// TIA Portal V17 export
// export: Created 2024-08-20T13:36:59.3159366Z, ExportSetting WithDefaults, DisplayName Totally Integrated Automation Portal, DisplayVersion V17 Update 4, DisplayName TIA Portal Openness, DisplayVersion V17 Update 4, DisplayName TIA Portal Version Control Interface, DisplayVersion V17, DisplayName STEP 7 Professional, DisplayVersion V17 Update 4, DisplayName STEP 7 Safety, DisplayVersion V17, DisplayName WinCC Advanced, DisplayVersion V17 Update 4
FUNCTION_BLOCK "ROD4"   // FB200, LAD
TITLE = Rodízio de 4 grupos
{ S7_Optimized_Access := 'FALSE' }
VERSION : 0.1
// stored: AutoNumber false, IsIECCheckEnabled false, SetENOAutomatically false, UDAEnableTagReadback false
   VAR_INPUT
      G1OK : Bool;   // GRUPO EM CONDIÇÕES DE OPERAÇÃO
      G2OK : Bool;   // GRUPO EM CONDIÇÕES DE OPERAÇÃO
      G3OK : Bool;   // GRUPO EM CONDIÇÕES DE OPERAÇÃO
      G4OK : Bool;   // GRUPO EM CONDIÇÕES DE OPERAÇÃO
      G1L : Bool;   // GRUPO LIGADO
      G2L : Bool;   // GRUPO LIGADO
      G3L : Bool;   // GRUPO LIGADO
      G4L : Bool;   // GRUPO LIGADO
      TEROD : DInt;   // TEMPOPARA RODÍZIO DAS BOMBAS
      LIGP : Bool;   // LIGA BOMBA PRINCIPAL
      LIGC1 : Bool;   // LIGA BOMBA COMPLEMENTAR 1
      LIGC2 : Bool;   // LIGA BOMBA COMPLEMENTAR 2
      LIGC3 : Bool;   // LIGA BOMBA COMPLEMENTAR 3
      DESAB : Bool;   // DESABILITA FUNCIONAMENTO DOS GRUPOS
      T1S : Bool;   // PULSO A CADA 1 SEGUNDO
   END_VAR
   VAR_OUTPUT
      G1P : Bool;   // GRUPO 1 SELECIONADO COMO PRINCIPAL
      G2P : Bool;   // GRUPO 2 SELECIONADO COMO PRINCIPAL
      G3P : Bool;   // GRUPO 3 SELECIONADO COMO PRINCIPAL
      G4P : Bool;   // GRUPO 4 SELECIONADO COMO PRINCIPAL
      G1C1 : Bool;   // GRUPO 1 SELECIONADO COMO COMPLEMENTAR 1
      G2C1 : Bool;   // GRUPO 2 SELECIONADO COMO COMPLEMENTAR 1
      G3C1 : Bool;   // GRUPO 3 SELECIONADO COMO COMPLEMENTAR 1
      G4C1 : Bool;   // GRUPO 4 SELECIONADO COMO COMPLEMENTAR 1
      G1C2 : Bool;   // GRUPO 1 SELECIONADO COMO COMPLEMENTAR 2
      G2C2 : Bool;   // GRUPO 2 SELECIONADO COMO COMPLEMENTAR 2
      G3C2 : Bool;   // GRUPO 3 SELECIONADO COMO COMPLEMENTAR 3
      G4C2 : Bool;   // GRUPO 4 SELECIONADO COMO COMPLEMENTAR 4
      G1C3 : Bool;   // GRUPO 1 SELECIONADO COMO COMPLEMENTAR 3
      G2C3 : Bool;   // GRUPO 2 SELECIONADO COMO COMPLEMENTAR 3
      G3C3 : Bool;   // GRUPO 3 SELECIONADO COMO COMPLEMENTAR 3
      G4C3 : Bool;   // GRUPO 4 SELECIONADO COMO COMPLEMENTAR 3
      LG1 : Bool;   // LIGA GRUPO 1
      LG2 : Bool;   // LIGA GRUPO 2
      LG3 : Bool;   // LIGA GRUPO 3
      LG4 : Bool;   // LIGA GRUPO 4
   END_VAR
   VAR_IN_OUT
      TOG1P : DInt;   // TEMPO DE OPERAÇÃO GRUPO 1
      TOG2P : DInt;   // TEMPO DE OPERAÇÃO GRUPO 2
      TOG3P : DInt;   // TEMPO DE OPERAÇÃO GRUPO 3
      TOG4P : DInt;   // TEMPO DE OPERAÇÃO GRUPO 4
      TEOKG1 : Real;   // TEMPO OK GRUPO 1
      TEOKG2 : Real;   // TEMPO OK GRUPO 2
      TEOKG3 : Real;   // TEMPO OK GRUPO 3
      TEOKG4 : Real;   // TEMPO OK GRUPO 4
   END_VAR
   VAR DB_SPECIFIC
      GR1SELP : Bool;   // SELECIONADO COMO PRINCIPAL
      GR2SELP : Bool;   // SELECIONADO COMO PRINCIPAL
      GR3SELP : Bool;   // SELECIONADO COMO PRINCIPAL
      GR4SELP : Bool;   // SELECIONADO COMO PRINCIPAL
      GR1SELC1 : Bool;   // SELECIONADO COMO COMPLEMENTAR 1
      GR2SELC1 : Bool;   // SELECIONADO COMO COMPLEMENTAR 1
      GR3SELC1 : Bool;   // SELECIONADO COMO COMPLEMENTAR 1
      GR4SELC1 : Bool;   // SELECIONADO COMO COMPLEMENTAR 1
      GR1SELC2 : Bool;   // SELECIONADO COMO COMPLEMENTAR 2
      GR2SELC2 : Bool;   // SELECIONADO COMO COMPLEMENTAR 2
      GR3SELC2 : Bool;   // SELECIONADO COMO COMPLEMENTAR 2
      GR4SELC2 : Bool;   // SELECIONADO COMO COMPLEMENTAR 2
      GR1SELC3 : Bool;   // SELECIONADO COMO COMPLEMENTAR 3
      GR2SELC3 : Bool;   // SELECIONADO COMO COMPLEMENTAR 3
      GR3SELC3 : Bool;   // SELECIONADO COMO COMPLEMENTAR 3
      GR4SELC3 : Bool;   // SELECIONADO COMO COMPLEMENTAR 3
      PS1SG1 : Bool;   // AUXILIAR DE PULSO
      PS1SG2 : Bool;   // AUXILIAR DE PULSO
      PS1SG3 : Bool;   // AUXILIAR DE PULSO
      PS1SG4 : Bool;   // AUXILIAR DE PULSO
      PS1 : Bool;   // AUXILIAR DE PULSO
      PS2 : Bool;   // AUXILIAR DE PULSO
      PS3 : Bool;   // AUXILIAR DE PULSO
      PS4 : Bool;   // AUXILIAR DE PULSO
      FIMTEG1 : Bool;   // FIM DO TEMPO DE EXISTÊNCIA DO GRUPO 1
      FIMTEG2 : Bool;   // FIM DO TEMPO DE EXISTÊNCIA DO GRUPO 2
      FIMTEG3 : Bool;   // FIM DO TEMPO DE EXISTÊNCIA DO GRUPO 3
      FIMTEG4 : Bool;   // FIM DO TEMPO DE EXISTÊNCIA DO GRUPO 4
      SDESG1 : Bool;   // SOLICITAÇÃO DE DESLIGAMENTO
      SDESG2 : Bool;   // SOLICITAÇÃO DE DESLIGAMENTO
      SDESG3 : Bool;   // SOLICITAÇÃO DE DESLIGAMENTO
      SDESG4 : Bool;   // SOLICITAÇÃO DE DESLIGAMENTO
      GPL : Bool;   // GRUPO PRINCIPAL LIGADO
      GC1L : Bool;   // GRUPO COMPLEMENTAR 1 LIGADO
      GC2L : Bool;   // GRUPO COMPLEMENTAR 2 LIGADO
      GC3L : Bool;   // GRUPO COMPLEMENTAR 3 LIGADO
      SO_L : Bool;   // SOLICITAÇÃO DE PARTIDA
      SO_D : Bool;   // SOLICITAÇÃO DE DESLIGAMENTO
      RTEOKG1 : Bool;   // RESET TEMPO OK
      RTEOKG2 : Bool;   // RESET TEMPO OK
      RTEOKG3 : Bool;   // RESET TEMPO OK
      RTEOKG4 : Bool;   // RESET TEMPO OK
      TON1 { S7_SetPoint := 'True'} : TON_TIME;   // TEMPORIZADOR
      TON2 { S7_SetPoint := 'True'} : TON_TIME;   // TEMPORIZADOR
      TON3 { S7_SetPoint := 'True'} : TON_TIME;   // TEMPORIZADOR
      TON4 { S7_SetPoint := 'True'} : TON_TIME;   // TEMPORIZADOR
      TSDG1 { S7_SetPoint := 'True'} : TON_TIME;   // TEMPORIZADOR
      TSDG2 { S7_SetPoint := 'True'} : TON_TIME;   // TEMPORIZADOR
      TSDG3 { S7_SetPoint := 'True'} : TON_TIME;   // TEMPORIZADOR
      TSDG4 { S7_SetPoint := 'True'} : TON_TIME;   // TEMPORIZADOR
   END_VAR
   VAR_TEMP
      PRI12 : Bool;   // PRIORIDADE GRUPO 1
      PRI13 : Bool;   // PRIORIDADE GRUPO 1
      PRI14 : Bool;   // PRIORIDADE GRUPO 1
      PRI23 : Bool;   // PRIORIDADE GRUPO 2
      PRI24 : Bool;   // PRIORIDADE GRUPO 2
      PRI34 : Bool;   // PRIORIDADE GRUPO 3
      TMROD : Real;   // TEMPO DE RODIZIO
      NGS : Int;   // NÚMERO DE GRUPOS SOLICITADOS
      NGF : Int;   // NÚMERO DE GRUPOS FUNCIONANDO
      AUX01 : Int;   // AUXILIAR UTILIZADO NA LÓGICA
      AUX02 : Int;   // AUXILIAR UTILIZADO NA LÓGICA
      AUX03 : Int;   // AUXILIAR UTILIZADO NA LÓGICA
      AUX04 : Int;   // AUXILIAR UTILIZADO NA LÓGICA
      AUX05 : Bool;   // AUXILIAR UTILIZADO NA LÓGICA
      AUX06 : Bool;   // AUXILIAR UTILIZADO NA LÓGICA
      AUX07 : Bool;   // AUXILIAR UTILIZADO NA LÓGICA
      AUX08 : Bool;   // AUXILIAR UTILIZADO NA LÓGICA
      ETT1 : Time;   // EFETIVO DO TEMPORIZADOR
      ETT2 : Time;   // EFETIVO DO TEMPORIZADOR
      ETT3 : Time;   // EFETIVO DO TEMPORIZADOR
      ETT4 : Time;   // EFETIVO DO TEMPORIZADOR
      ETTSDG4 : Time;   // EFETIVO DO TEMPORIZADOR
      ETTSDG3 : Time;   // EFETIVO DO TEMPORIZADOR
      ETTSDG2 : Time;   // EFETIVO DO TEMPORIZADOR
      ETTSDG1 : Time;   // EFETIVO DO TEMPORIZADOR
   END_VAR
   VAR_TEMP   // added for the SCL form of the ladder/FBD networks
      _w1 : Bool;
   END_VAR
BEGIN

REGION Network 1: Tranforme em segundo o tempo de rodízio dos sopradores
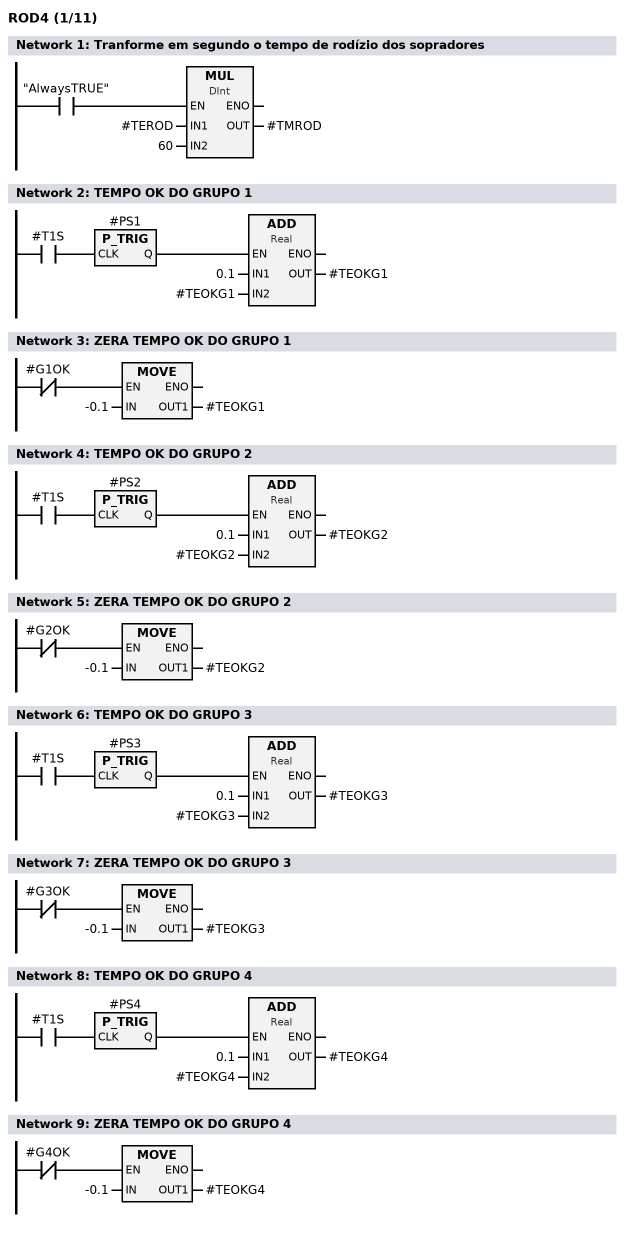
   RUNG wire#powerrail
      Contact( "AlwaysTRUE" )
      { S7_Templates := "SrcType := DInt"; S7_GenerateENO := "TRUE" } Mul(in1 := #TEROD, in2 := 60, out => #TMROD)
   END_RUNG
   // the same network as SCL:
   IF "AlwaysTRUE" THEN #TMROD := #TEROD * 60; END_IF;
END_REGION

REGION Network 2: TEMPO OK DO GRUPO 1
   RUNG wire#powerrail
      Contact( #T1S )
      P_Trig( #PS1 )
      { S7_Templates := "SrcType := Real"; S7_GenerateENO := "TRUE" } Add(in1 := 0.1, in2 := #TEOKG1, out => #TEOKG1)
   END_RUNG
   // the same network as SCL:
   #_w1 := #T1S AND NOT #PS1;   // rising edge
   #PS1 := #T1S;
   IF #_w1 THEN #TEOKG1 := 0.1 + #TEOKG1; END_IF;
END_REGION

REGION Network 3: ZERA TEMPO OK DO GRUPO 1
   RUNG wire#powerrail
      I_Contact( #G1OK )
      { S7_GenerateENO := "TRUE" } Move(in := -0.1, out1 => #TEOKG1)
   END_RUNG
   // the same network as SCL:
   IF NOT #G1OK THEN #TEOKG1 := -0.1; END_IF;
END_REGION

REGION Network 4: TEMPO OK DO GRUPO 2
   RUNG wire#powerrail
      Contact( #T1S )
      P_Trig( #PS2 )
      { S7_Templates := "SrcType := Real"; S7_GenerateENO := "TRUE" } Add(in1 := 0.1, in2 := #TEOKG2, out => #TEOKG2)
   END_RUNG
   // the same network as SCL:
   #_w1 := #T1S AND NOT #PS2;   // rising edge
   #PS2 := #T1S;
   IF #_w1 THEN #TEOKG2 := 0.1 + #TEOKG2; END_IF;
END_REGION

REGION Network 5: ZERA TEMPO OK DO GRUPO 2
   RUNG wire#powerrail
      I_Contact( #G2OK )
      { S7_GenerateENO := "TRUE" } Move(in := -0.1, out1 => #TEOKG2)
   END_RUNG
   // the same network as SCL:
   IF NOT #G2OK THEN #TEOKG2 := -0.1; END_IF;
END_REGION

REGION Network 6: TEMPO OK DO GRUPO 3
   RUNG wire#powerrail
      Contact( #T1S )
      P_Trig( #PS3 )
      { S7_Templates := "SrcType := Real"; S7_GenerateENO := "TRUE" } Add(in1 := 0.1, in2 := #TEOKG3, out => #TEOKG3)
   END_RUNG
   // the same network as SCL:
   #_w1 := #T1S AND NOT #PS3;   // rising edge
   #PS3 := #T1S;
   IF #_w1 THEN #TEOKG3 := 0.1 + #TEOKG3; END_IF;
END_REGION

REGION Network 7: ZERA TEMPO OK DO GRUPO 3
   RUNG wire#powerrail
      I_Contact( #G3OK )
      { S7_GenerateENO := "TRUE" } Move(in := -0.1, out1 => #TEOKG3)
   END_RUNG
   // the same network as SCL:
   IF NOT #G3OK THEN #TEOKG3 := -0.1; END_IF;
END_REGION

REGION Network 8: TEMPO OK DO GRUPO 4
   RUNG wire#powerrail
      Contact( #T1S )
      P_Trig( #PS4 )
      { S7_Templates := "SrcType := Real"; S7_GenerateENO := "TRUE" } Add(in1 := 0.1, in2 := #TEOKG4, out => #TEOKG4)
   END_RUNG
   // the same network as SCL:
   #_w1 := #T1S AND NOT #PS4;   // rising edge
   #PS4 := #T1S;
   IF #_w1 THEN #TEOKG4 := 0.1 + #TEOKG4; END_IF;
END_REGION

REGION Network 9: ZERA TEMPO OK DO GRUPO 4
   RUNG wire#powerrail
      I_Contact( #G4OK )
      { S7_GenerateENO := "TRUE" } Move(in := -0.1, out1 => #TEOKG4)
   END_RUNG
   // the same network as SCL:
   IF NOT #G4OK THEN #TEOKG4 := -0.1; END_IF;
END_REGION

REGION Network 10: DEFINIÇÇÃO DE PRIORIDADE DO GRUPO 1
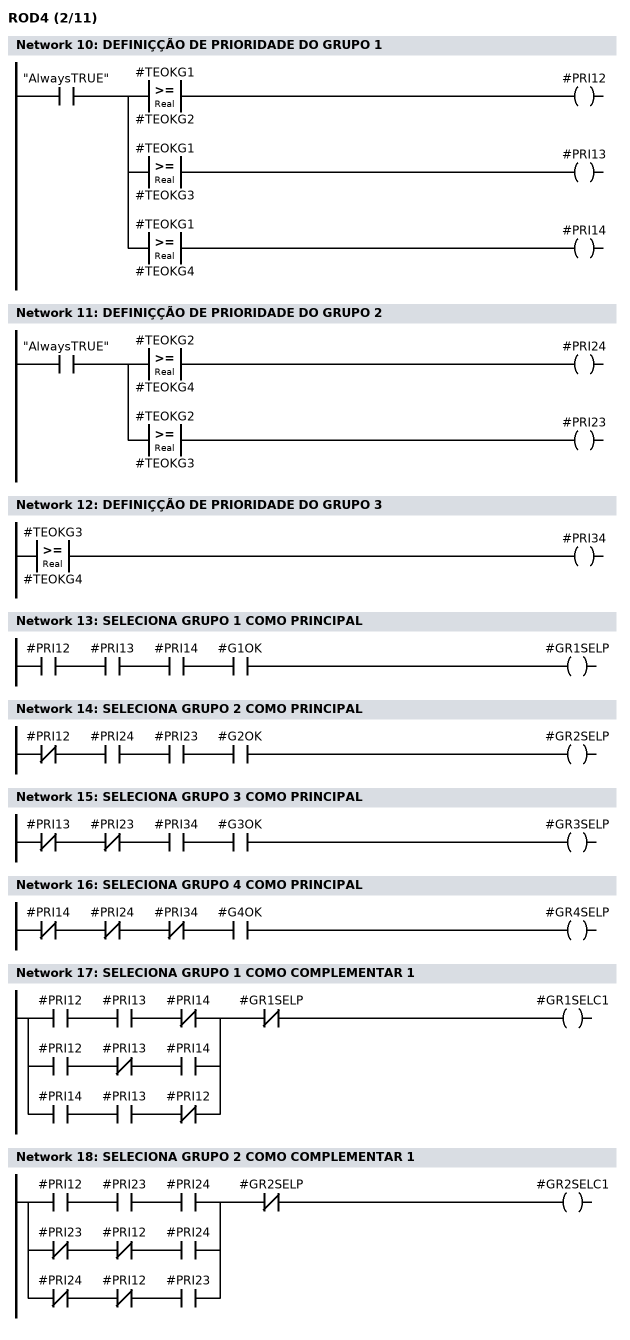
   RUNG wire#powerrail
      Contact( "AlwaysTRUE" )
      wire#w1
      { S7_Templates := "SrcType := Real" } GE_Contact(in1 := #TEOKG1, in2 := #TEOKG2)
      Coil( #PRI12 )
   END_RUNG
   RUNG wire#w1
      { S7_Templates := "SrcType := Real" } GE_Contact(in1 := #TEOKG1, in2 := #TEOKG3)
      Coil( #PRI13 )
   END_RUNG
   RUNG wire#w1
      { S7_Templates := "SrcType := Real" } GE_Contact(in1 := #TEOKG1, in2 := #TEOKG4)
      Coil( #PRI14 )
   END_RUNG
   // the same network as SCL:
   #PRI12 := "AlwaysTRUE" AND (#TEOKG1 >= #TEOKG2);
   #PRI13 := "AlwaysTRUE" AND (#TEOKG1 >= #TEOKG3);
   #PRI14 := "AlwaysTRUE" AND (#TEOKG1 >= #TEOKG4);
END_REGION

REGION Network 11: DEFINIÇÇÃO DE PRIORIDADE DO GRUPO 2
   RUNG wire#powerrail
      Contact( "AlwaysTRUE" )
      wire#w1
      { S7_Templates := "SrcType := Real" } GE_Contact(in1 := #TEOKG2, in2 := #TEOKG4)
      Coil( #PRI24 )
   END_RUNG
   RUNG wire#w1
      { S7_Templates := "SrcType := Real" } GE_Contact(in1 := #TEOKG2, in2 := #TEOKG3)
      Coil( #PRI23 )
   END_RUNG
   // the same network as SCL:
   #PRI24 := "AlwaysTRUE" AND (#TEOKG2 >= #TEOKG4);
   #PRI23 := "AlwaysTRUE" AND (#TEOKG2 >= #TEOKG3);
END_REGION

REGION Network 12: DEFINIÇÇÃO DE PRIORIDADE DO GRUPO 3
   RUNG wire#powerrail
      { S7_Templates := "SrcType := Real" } GE_Contact(in1 := #TEOKG3, in2 := #TEOKG4)
      Coil( #PRI34 )
   END_RUNG
   // the same network as SCL:
   #PRI34 := #TEOKG3 >= #TEOKG4;
END_REGION

REGION Network 13: SELECIONA GRUPO 1 COMO PRINCIPAL
   RUNG wire#powerrail
      Contact( #PRI12 )
      Contact( #PRI13 )
      Contact( #PRI14 )
      Contact( #G1OK )
      Coil( #GR1SELP )
   END_RUNG
   // the same network as SCL:
   #GR1SELP := #PRI12 AND #PRI13 AND #PRI14 AND #G1OK;
END_REGION

REGION Network 14: SELECIONA GRUPO 2 COMO PRINCIPAL
   RUNG wire#powerrail
      I_Contact( #PRI12 )
      Contact( #PRI24 )
      Contact( #PRI23 )
      Contact( #G2OK )
      Coil( #GR2SELP )
   END_RUNG
   // the same network as SCL:
   #GR2SELP := NOT #PRI12 AND #PRI24 AND #PRI23 AND #G2OK;
END_REGION

REGION Network 15: SELECIONA GRUPO 3 COMO PRINCIPAL
   RUNG wire#powerrail
      I_Contact( #PRI13 )
      I_Contact( #PRI23 )
      Contact( #PRI34 )
      Contact( #G3OK )
      Coil( #GR3SELP )
   END_RUNG
   // the same network as SCL:
   #GR3SELP := NOT #PRI13 AND NOT #PRI23 AND #PRI34 AND #G3OK;
END_REGION

REGION Network 16: SELECIONA GRUPO 4 COMO PRINCIPAL
   RUNG wire#powerrail
      I_Contact( #PRI14 )
      I_Contact( #PRI24 )
      I_Contact( #PRI34 )
      Contact( #G4OK )
      Coil( #GR4SELP )
   END_RUNG
   // the same network as SCL:
   #GR4SELP := NOT #PRI14 AND NOT #PRI24 AND NOT #PRI34 AND #G4OK;
END_REGION

REGION Network 17: SELECIONA GRUPO 1 COMO COMPLEMENTAR 1
   RUNG wire#powerrail
      Contact( #PRI12 )
      Contact( #PRI13 )
      I_Contact( #PRI14 )
      wire#w1
      I_Contact( #GR1SELP )
      Coil( #GR1SELC1 )
   END_RUNG
   RUNG wire#powerrail
      Contact( #PRI12 )
      I_Contact( #PRI13 )
      Contact( #PRI14 )
   END_RUNG wire#w1
   RUNG wire#powerrail
      Contact( #PRI14 )
      Contact( #PRI13 )
      I_Contact( #PRI12 )
   END_RUNG wire#w1
   // the same network as SCL:
   #GR1SELC1 := ((#PRI12 AND #PRI13 AND NOT #PRI14) OR (#PRI12 AND NOT #PRI13 AND #PRI14) OR (#PRI14 AND #PRI13 AND NOT #PRI12)) AND NOT #GR1SELP;
END_REGION

REGION Network 18: SELECIONA GRUPO 2 COMO COMPLEMENTAR 1
   RUNG wire#powerrail
      Contact( #PRI12 )
      Contact( #PRI23 )
      Contact( #PRI24 )
      wire#w1
      I_Contact( #GR2SELP )
      Coil( #GR2SELC1 )
   END_RUNG
   RUNG wire#powerrail
      I_Contact( #PRI23 )
      I_Contact( #PRI12 )
      Contact( #PRI24 )
   END_RUNG wire#w1
   RUNG wire#powerrail
      I_Contact( #PRI24 )
      I_Contact( #PRI12 )
      Contact( #PRI23 )
   END_RUNG wire#w1
   // the same network as SCL:
   #GR2SELC1 := ((#PRI12 AND #PRI23 AND #PRI24) OR (NOT #PRI23 AND NOT #PRI12 AND #PRI24) OR (NOT #PRI24 AND NOT #PRI12 AND #PRI23)) AND NOT #GR2SELP;
END_REGION

REGION Network 19: SELECIONA GRUPO 3 COMO COMPLEMENTAR 1
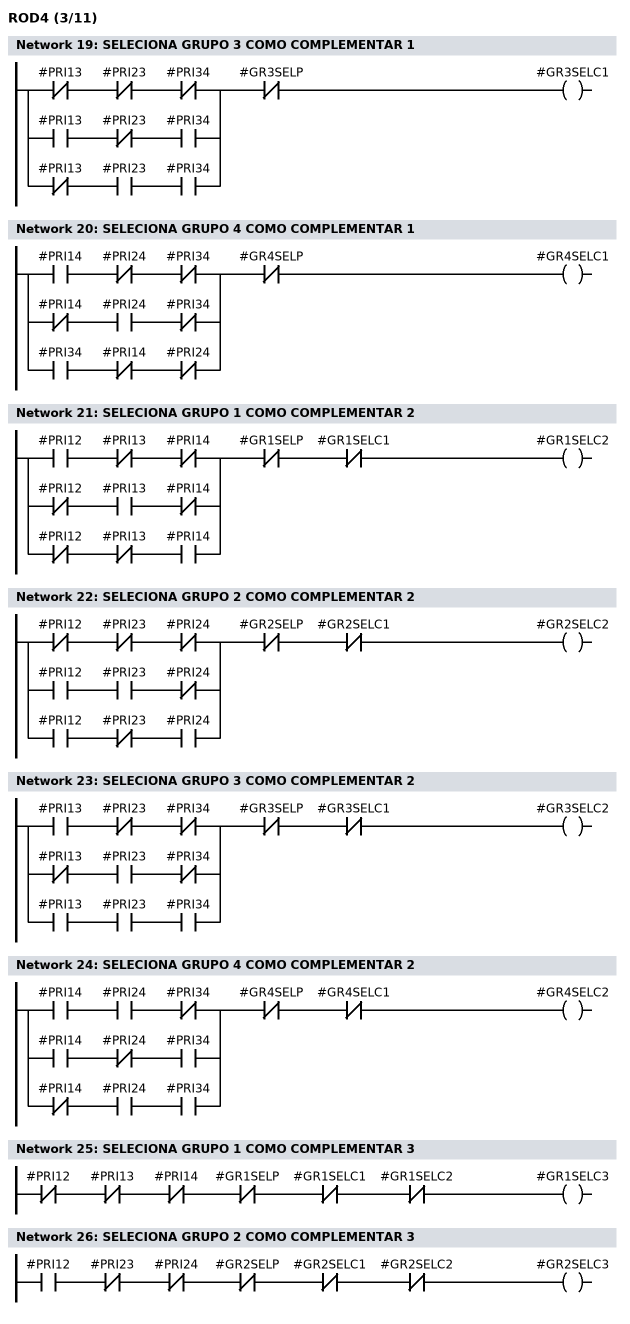
   RUNG wire#powerrail
      I_Contact( #PRI13 )
      I_Contact( #PRI23 )
      I_Contact( #PRI34 )
      wire#w1
      I_Contact( #GR3SELP )
      Coil( #GR3SELC1 )
   END_RUNG
   RUNG wire#powerrail
      Contact( #PRI13 )
      I_Contact( #PRI23 )
      Contact( #PRI34 )
   END_RUNG wire#w1
   RUNG wire#powerrail
      I_Contact( #PRI13 )
      Contact( #PRI23 )
      Contact( #PRI34 )
   END_RUNG wire#w1
   // the same network as SCL:
   #GR3SELC1 := ((NOT #PRI13 AND NOT #PRI23 AND NOT #PRI34) OR (#PRI13 AND NOT #PRI23 AND #PRI34) OR (NOT #PRI13 AND #PRI23 AND #PRI34)) AND NOT #GR3SELP;
END_REGION

REGION Network 20: SELECIONA GRUPO 4 COMO COMPLEMENTAR 1
   RUNG wire#powerrail
      Contact( #PRI14 )
      I_Contact( #PRI24 )
      I_Contact( #PRI34 )
      wire#w1
      I_Contact( #GR4SELP )
      Coil( #GR4SELC1 )
   END_RUNG
   RUNG wire#powerrail
      I_Contact( #PRI14 )
      Contact( #PRI24 )
      I_Contact( #PRI34 )
   END_RUNG wire#w1
   RUNG wire#powerrail
      Contact( #PRI34 )
      I_Contact( #PRI14 )
      I_Contact( #PRI24 )
   END_RUNG wire#w1
   // the same network as SCL:
   #GR4SELC1 := ((#PRI14 AND NOT #PRI24 AND NOT #PRI34) OR (NOT #PRI14 AND #PRI24 AND NOT #PRI34) OR (#PRI34 AND NOT #PRI14 AND NOT #PRI24)) AND NOT #GR4SELP;
END_REGION

REGION Network 21: SELECIONA GRUPO 1 COMO COMPLEMENTAR 2
   RUNG wire#powerrail
      Contact( #PRI12 )
      I_Contact( #PRI13 )
      I_Contact( #PRI14 )
      wire#w1
      I_Contact( #GR1SELP )
      I_Contact( #GR1SELC1 )
      Coil( #GR1SELC2 )
   END_RUNG
   RUNG wire#powerrail
      I_Contact( #PRI12 )
      Contact( #PRI13 )
      I_Contact( #PRI14 )
   END_RUNG wire#w1
   RUNG wire#powerrail
      I_Contact( #PRI12 )
      I_Contact( #PRI13 )
      Contact( #PRI14 )
   END_RUNG wire#w1
   // the same network as SCL:
   #GR1SELC2 := ((#PRI12 AND NOT #PRI13 AND NOT #PRI14) OR (NOT #PRI12 AND #PRI13 AND NOT #PRI14) OR (NOT #PRI12 AND NOT #PRI13 AND #PRI14)) AND NOT #GR1SELP AND NOT #GR1SELC1;
END_REGION

REGION Network 22: SELECIONA GRUPO 2 COMO COMPLEMENTAR 2
   RUNG wire#powerrail
      I_Contact( #PRI12 )
      I_Contact( #PRI23 )
      I_Contact( #PRI24 )
      wire#w1
      I_Contact( #GR2SELP )
      I_Contact( #GR2SELC1 )
      Coil( #GR2SELC2 )
   END_RUNG
   RUNG wire#powerrail
      Contact( #PRI12 )
      Contact( #PRI23 )
      I_Contact( #PRI24 )
   END_RUNG wire#w1
   RUNG wire#powerrail
      Contact( #PRI12 )
      I_Contact( #PRI23 )
      Contact( #PRI24 )
   END_RUNG wire#w1
   // the same network as SCL:
   #GR2SELC2 := ((NOT #PRI12 AND NOT #PRI23 AND NOT #PRI24) OR (#PRI12 AND #PRI23 AND NOT #PRI24) OR (#PRI12 AND NOT #PRI23 AND #PRI24)) AND NOT #GR2SELP AND NOT #GR2SELC1;
END_REGION

REGION Network 23: SELECIONA GRUPO 3 COMO COMPLEMENTAR 2
   RUNG wire#powerrail
      Contact( #PRI13 )
      I_Contact( #PRI23 )
      I_Contact( #PRI34 )
      wire#w1
      I_Contact( #GR3SELP )
      I_Contact( #GR3SELC1 )
      Coil( #GR3SELC2 )
   END_RUNG
   RUNG wire#powerrail
      I_Contact( #PRI13 )
      Contact( #PRI23 )
      I_Contact( #PRI34 )
   END_RUNG wire#w1
   RUNG wire#powerrail
      Contact( #PRI13 )
      Contact( #PRI23 )
      Contact( #PRI34 )
   END_RUNG wire#w1
   // the same network as SCL:
   #GR3SELC2 := ((#PRI13 AND NOT #PRI23 AND NOT #PRI34) OR (NOT #PRI13 AND #PRI23 AND NOT #PRI34) OR (#PRI13 AND #PRI23 AND #PRI34)) AND NOT #GR3SELP AND NOT #GR3SELC1;
END_REGION

REGION Network 24: SELECIONA GRUPO 4 COMO COMPLEMENTAR 2
   RUNG wire#powerrail
      Contact( #PRI14 )
      Contact( #PRI24 )
      I_Contact( #PRI34 )
      wire#w1
      I_Contact( #GR4SELP )
      I_Contact( #GR4SELC1 )
      Coil( #GR4SELC2 )
   END_RUNG
   RUNG wire#powerrail
      Contact( #PRI14 )
      I_Contact( #PRI24 )
      Contact( #PRI34 )
   END_RUNG wire#w1
   RUNG wire#powerrail
      I_Contact( #PRI14 )
      Contact( #PRI24 )
      Contact( #PRI34 )
   END_RUNG wire#w1
   // the same network as SCL:
   #GR4SELC2 := ((#PRI14 AND #PRI24 AND NOT #PRI34) OR (#PRI14 AND NOT #PRI24 AND #PRI34) OR (NOT #PRI14 AND #PRI24 AND #PRI34)) AND NOT #GR4SELP AND NOT #GR4SELC1;
END_REGION

REGION Network 25: SELECIONA GRUPO 1 COMO COMPLEMENTAR 3
   RUNG wire#powerrail
      I_Contact( #PRI12 )
      I_Contact( #PRI13 )
      I_Contact( #PRI14 )
      I_Contact( #GR1SELP )
      I_Contact( #GR1SELC1 )
      I_Contact( #GR1SELC2 )
      Coil( #GR1SELC3 )
   END_RUNG
   // the same network as SCL:
   #GR1SELC3 := NOT #PRI12 AND NOT #PRI13 AND NOT #PRI14 AND NOT #GR1SELP AND NOT #GR1SELC1 AND NOT #GR1SELC2;
END_REGION

REGION Network 26: SELECIONA GRUPO 2 COMO COMPLEMENTAR 3
   RUNG wire#powerrail
      Contact( #PRI12 )
      I_Contact( #PRI23 )
      I_Contact( #PRI24 )
      I_Contact( #GR2SELP )
      I_Contact( #GR2SELC1 )
      I_Contact( #GR2SELC2 )
      Coil( #GR2SELC3 )
   END_RUNG
   // the same network as SCL:
   #GR2SELC3 := #PRI12 AND NOT #PRI23 AND NOT #PRI24 AND NOT #GR2SELP AND NOT #GR2SELC1 AND NOT #GR2SELC2;
END_REGION

REGION Network 27: SELECIONA GRUPO 3 COMO COMPLEMENTAR 3
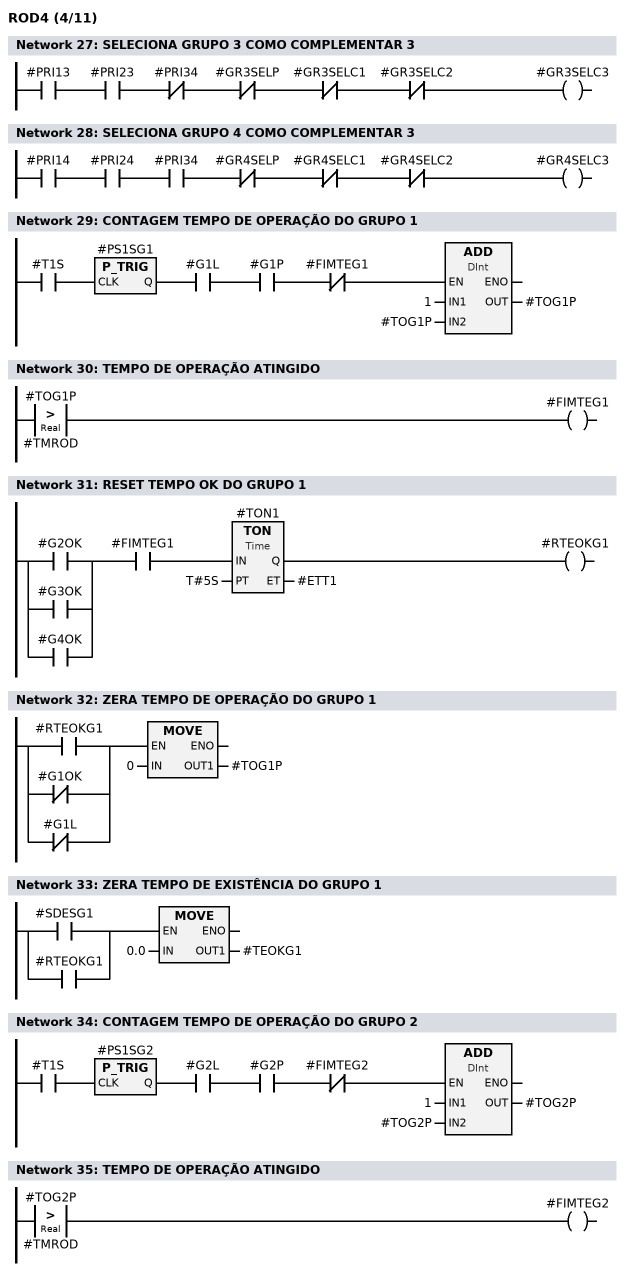
   RUNG wire#powerrail
      Contact( #PRI13 )
      Contact( #PRI23 )
      I_Contact( #PRI34 )
      I_Contact( #GR3SELP )
      I_Contact( #GR3SELC1 )
      I_Contact( #GR3SELC2 )
      Coil( #GR3SELC3 )
   END_RUNG
   // the same network as SCL:
   #GR3SELC3 := #PRI13 AND #PRI23 AND NOT #PRI34 AND NOT #GR3SELP AND NOT #GR3SELC1 AND NOT #GR3SELC2;
END_REGION

REGION Network 28: SELECIONA GRUPO 4 COMO COMPLEMENTAR 3
   RUNG wire#powerrail
      Contact( #PRI14 )
      Contact( #PRI24 )
      Contact( #PRI34 )
      I_Contact( #GR4SELP )
      I_Contact( #GR4SELC1 )
      I_Contact( #GR4SELC2 )
      Coil( #GR4SELC3 )
   END_RUNG
   // the same network as SCL:
   #GR4SELC3 := #PRI14 AND #PRI24 AND #PRI34 AND NOT #GR4SELP AND NOT #GR4SELC1 AND NOT #GR4SELC2;
END_REGION

REGION Network 29: CONTAGEM TEMPO DE OPERAÇÃO DO GRUPO 1
   RUNG wire#powerrail
      Contact( #T1S )
      P_Trig( #PS1SG1 )
      Contact( #G1L )
      Contact( #G1P )
      I_Contact( #FIMTEG1 )
      { S7_Templates := "SrcType := DInt"; S7_GenerateENO := "TRUE" } Add(in1 := 1, in2 := #TOG1P, out => #TOG1P)
   END_RUNG
   // the same network as SCL:
   #_w1 := #T1S AND NOT #PS1SG1;   // rising edge
   #PS1SG1 := #T1S;
   IF #_w1 AND #G1L AND #G1P AND NOT #FIMTEG1 THEN #TOG1P := 1 + #TOG1P; END_IF;
END_REGION

REGION Network 30: TEMPO DE OPERAÇÃO ATINGIDO
   RUNG wire#powerrail
      { S7_Templates := "SrcType := Real" } GT_Contact(in1 := #TOG1P, in2 := #TMROD)
      Coil( #FIMTEG1 )
   END_RUNG
   // the same network as SCL:
   #FIMTEG1 := #TOG1P > #TMROD;
END_REGION

REGION Network 31: RESET TEMPO OK DO GRUPO 1
   RUNG wire#powerrail
      Contact( #G2OK )
      wire#w1
      Contact( #FIMTEG1 )
      { S7_Templates := "time_type := Time" } #TON1.TON(pt := T#5S, et => #ETT1)
      Coil( #RTEOKG1 )
   END_RUNG
   RUNG wire#powerrail
      Contact( #G3OK )
   END_RUNG wire#w1
   RUNG wire#powerrail
      Contact( #G4OK )
   END_RUNG wire#w1
   // the same network as SCL:
   #TON1(IN := (#G2OK OR #G3OK OR #G4OK) AND #FIMTEG1, PT := T#5S, ET => #ETT1);   // TON
   #RTEOKG1 := #TON1.Q;
END_REGION

REGION Network 32: ZERA TEMPO DE OPERAÇÃO DO GRUPO 1
   RUNG wire#powerrail
      Contact( #RTEOKG1 )
      wire#w1
      { S7_GenerateENO := "TRUE" } Move(in := 0, out1 => #TOG1P)
   END_RUNG
   RUNG wire#powerrail
      I_Contact( #G1OK )
   END_RUNG wire#w1
   RUNG wire#powerrail
      I_Contact( #G1L )
   END_RUNG wire#w1
   // the same network as SCL:
   IF #RTEOKG1 OR NOT #G1OK OR NOT #G1L THEN #TOG1P := 0; END_IF;
END_REGION

REGION Network 33: ZERA TEMPO DE EXISTÊNCIA DO GRUPO 1
   RUNG wire#powerrail
      Contact( #SDESG1 )
      wire#w1
      { S7_GenerateENO := "TRUE" } Move(in := 0.0, out1 => #TEOKG1)
   END_RUNG
   RUNG wire#powerrail
      Contact( #RTEOKG1 )
   END_RUNG wire#w1
   // the same network as SCL:
   IF #SDESG1 OR #RTEOKG1 THEN #TEOKG1 := 0.0; END_IF;
END_REGION

REGION Network 34: CONTAGEM TEMPO DE OPERAÇÃO DO GRUPO 2
   RUNG wire#powerrail
      Contact( #T1S )
      P_Trig( #PS1SG2 )
      Contact( #G2L )
      Contact( #G2P )
      I_Contact( #FIMTEG2 )
      { S7_Templates := "SrcType := DInt"; S7_GenerateENO := "TRUE" } Add(in1 := 1, in2 := #TOG2P, out => #TOG2P)
   END_RUNG
   // the same network as SCL:
   #_w1 := #T1S AND NOT #PS1SG2;   // rising edge
   #PS1SG2 := #T1S;
   IF #_w1 AND #G2L AND #G2P AND NOT #FIMTEG2 THEN #TOG2P := 1 + #TOG2P; END_IF;
END_REGION

REGION Network 35: TEMPO DE OPERAÇÃO ATINGIDO
   RUNG wire#powerrail
      { S7_Templates := "SrcType := Real" } GT_Contact(in1 := #TOG2P, in2 := #TMROD)
      Coil( #FIMTEG2 )
   END_RUNG
   // the same network as SCL:
   #FIMTEG2 := #TOG2P > #TMROD;
END_REGION

REGION Network 36: RESET TEMPO OK DO GRUPO 2
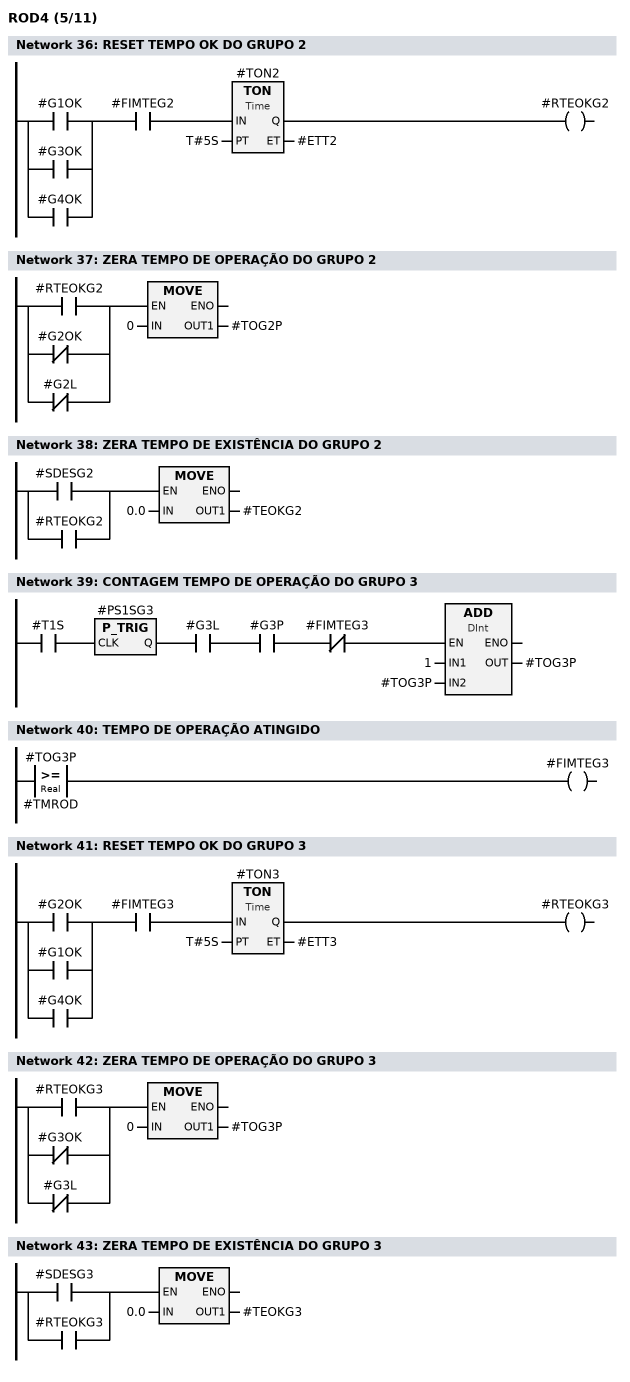
   RUNG wire#powerrail
      Contact( #G1OK )
      wire#w1
      Contact( #FIMTEG2 )
      { S7_Templates := "time_type := Time" } #TON2.TON(pt := T#5S, et => #ETT2)
      Coil( #RTEOKG2 )
   END_RUNG
   RUNG wire#powerrail
      Contact( #G3OK )
   END_RUNG wire#w1
   RUNG wire#powerrail
      Contact( #G4OK )
   END_RUNG wire#w1
   // the same network as SCL:
   #TON2(IN := (#G1OK OR #G3OK OR #G4OK) AND #FIMTEG2, PT := T#5S, ET => #ETT2);   // TON
   #RTEOKG2 := #TON2.Q;
END_REGION

REGION Network 37: ZERA TEMPO DE OPERAÇÃO DO GRUPO 2
   RUNG wire#powerrail
      Contact( #RTEOKG2 )
      wire#w1
      { S7_GenerateENO := "TRUE" } Move(in := 0, out1 => #TOG2P)
   END_RUNG
   RUNG wire#powerrail
      I_Contact( #G2OK )
   END_RUNG wire#w1
   RUNG wire#powerrail
      I_Contact( #G2L )
   END_RUNG wire#w1
   // the same network as SCL:
   IF #RTEOKG2 OR NOT #G2OK OR NOT #G2L THEN #TOG2P := 0; END_IF;
END_REGION

REGION Network 38: ZERA TEMPO DE EXISTÊNCIA DO GRUPO 2
   RUNG wire#powerrail
      Contact( #SDESG2 )
      wire#w1
      { S7_GenerateENO := "TRUE" } Move(in := 0.0, out1 => #TEOKG2)
   END_RUNG
   RUNG wire#powerrail
      Contact( #RTEOKG2 )
   END_RUNG wire#w1
   // the same network as SCL:
   IF #SDESG2 OR #RTEOKG2 THEN #TEOKG2 := 0.0; END_IF;
END_REGION

REGION Network 39: CONTAGEM TEMPO DE OPERAÇÃO DO GRUPO 3
   RUNG wire#powerrail
      Contact( #T1S )
      P_Trig( #PS1SG3 )
      Contact( #G3L )
      Contact( #G3P )
      I_Contact( #FIMTEG3 )
      { S7_Templates := "SrcType := DInt"; S7_GenerateENO := "TRUE" } Add(in1 := 1, in2 := #TOG3P, out => #TOG3P)
   END_RUNG
   // the same network as SCL:
   #_w1 := #T1S AND NOT #PS1SG3;   // rising edge
   #PS1SG3 := #T1S;
   IF #_w1 AND #G3L AND #G3P AND NOT #FIMTEG3 THEN #TOG3P := 1 + #TOG3P; END_IF;
END_REGION

REGION Network 40: TEMPO DE OPERAÇÃO ATINGIDO
   RUNG wire#powerrail
      { S7_Templates := "SrcType := Real" } GE_Contact(in1 := #TOG3P, in2 := #TMROD)
      Coil( #FIMTEG3 )
   END_RUNG
   // the same network as SCL:
   #FIMTEG3 := #TOG3P >= #TMROD;
END_REGION

REGION Network 41: RESET TEMPO OK DO GRUPO 3
   RUNG wire#powerrail
      Contact( #G2OK )
      wire#w1
      Contact( #FIMTEG3 )
      { S7_Templates := "time_type := Time" } #TON3.TON(pt := T#5S, et => #ETT3)
      Coil( #RTEOKG3 )
   END_RUNG
   RUNG wire#powerrail
      Contact( #G1OK )
   END_RUNG wire#w1
   RUNG wire#powerrail
      Contact( #G4OK )
   END_RUNG wire#w1
   // the same network as SCL:
   #TON3(IN := (#G2OK OR #G1OK OR #G4OK) AND #FIMTEG3, PT := T#5S, ET => #ETT3);   // TON
   #RTEOKG3 := #TON3.Q;
END_REGION

REGION Network 42: ZERA TEMPO DE OPERAÇÃO DO GRUPO 3
   RUNG wire#powerrail
      Contact( #RTEOKG3 )
      wire#w1
      { S7_GenerateENO := "TRUE" } Move(in := 0, out1 => #TOG3P)
   END_RUNG
   RUNG wire#powerrail
      I_Contact( #G3OK )
   END_RUNG wire#w1
   RUNG wire#powerrail
      I_Contact( #G3L )
   END_RUNG wire#w1
   // the same network as SCL:
   IF #RTEOKG3 OR NOT #G3OK OR NOT #G3L THEN #TOG3P := 0; END_IF;
END_REGION

REGION Network 43: ZERA TEMPO DE EXISTÊNCIA DO GRUPO 3
   RUNG wire#powerrail
      Contact( #SDESG3 )
      wire#w1
      { S7_GenerateENO := "TRUE" } Move(in := 0.0, out1 => #TEOKG3)
   END_RUNG
   RUNG wire#powerrail
      Contact( #RTEOKG3 )
   END_RUNG wire#w1
   // the same network as SCL:
   IF #SDESG3 OR #RTEOKG3 THEN #TEOKG3 := 0.0; END_IF;
END_REGION

REGION Network 44: CONTAGEM TEMPO DE OPERAÇÃO DO GRUPO 4
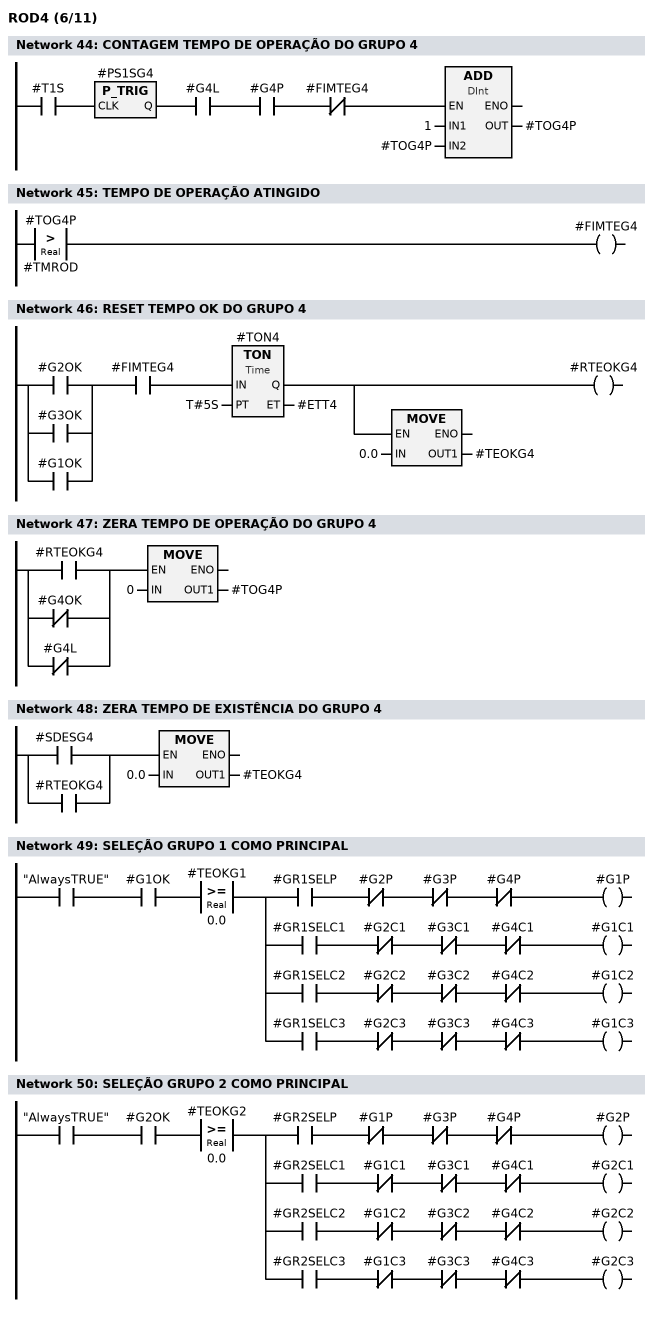
   RUNG wire#powerrail
      Contact( #T1S )
      P_Trig( #PS1SG4 )
      Contact( #G4L )
      Contact( #G4P )
      I_Contact( #FIMTEG4 )
      { S7_Templates := "SrcType := DInt"; S7_GenerateENO := "TRUE" } Add(in1 := 1, in2 := #TOG4P, out => #TOG4P)
   END_RUNG
   // the same network as SCL:
   #_w1 := #T1S AND NOT #PS1SG4;   // rising edge
   #PS1SG4 := #T1S;
   IF #_w1 AND #G4L AND #G4P AND NOT #FIMTEG4 THEN #TOG4P := 1 + #TOG4P; END_IF;
END_REGION

REGION Network 45: TEMPO DE OPERAÇÃO ATINGIDO
   RUNG wire#powerrail
      { S7_Templates := "SrcType := Real" } GT_Contact(in1 := #TOG4P, in2 := #TMROD)
      Coil( #FIMTEG4 )
   END_RUNG
   // the same network as SCL:
   #FIMTEG4 := #TOG4P > #TMROD;
END_REGION

REGION Network 46: RESET TEMPO OK DO GRUPO 4
   RUNG wire#powerrail
      Contact( #G2OK )
      wire#w1
      Contact( #FIMTEG4 )
      { S7_Templates := "time_type := Time" } #TON4.TON(pt := T#5S, et => #ETT4)
      wire#w2
      Coil( #RTEOKG4 )
   END_RUNG
   RUNG wire#powerrail
      Contact( #G3OK )
   END_RUNG wire#w1
   RUNG wire#powerrail
      Contact( #G1OK )
   END_RUNG wire#w1
   RUNG wire#w2
      { S7_GenerateENO := "TRUE" } Move(in := 0.0, out1 => #TEOKG4)
   END_RUNG
   // the same network as SCL:
   #TON4(IN := (#G2OK OR #G3OK OR #G1OK) AND #FIMTEG4, PT := T#5S, ET => #ETT4);   // TON
   #RTEOKG4 := #TON4.Q;
   IF #TON4.Q THEN #TEOKG4 := 0.0; END_IF;
END_REGION

REGION Network 47: ZERA TEMPO DE OPERAÇÃO DO GRUPO 4
   RUNG wire#powerrail
      Contact( #RTEOKG4 )
      wire#w1
      { S7_GenerateENO := "TRUE" } Move(in := 0, out1 => #TOG4P)
   END_RUNG
   RUNG wire#powerrail
      I_Contact( #G4OK )
   END_RUNG wire#w1
   RUNG wire#powerrail
      I_Contact( #G4L )
   END_RUNG wire#w1
   // the same network as SCL:
   IF #RTEOKG4 OR NOT #G4OK OR NOT #G4L THEN #TOG4P := 0; END_IF;
END_REGION

REGION Network 48: ZERA TEMPO DE EXISTÊNCIA DO GRUPO 4
   RUNG wire#powerrail
      Contact( #SDESG4 )
      wire#w1
      { S7_GenerateENO := "TRUE" } Move(in := 0.0, out1 => #TEOKG4)
   END_RUNG
   RUNG wire#powerrail
      Contact( #RTEOKG4 )
   END_RUNG wire#w1
   // the same network as SCL:
   IF #SDESG4 OR #RTEOKG4 THEN #TEOKG4 := 0.0; END_IF;
END_REGION

REGION Network 49: SELEÇÃO GRUPO 1 COMO PRINCIPAL
   RUNG wire#powerrail
      Contact( "AlwaysTRUE" )
      Contact( #G1OK )
      { S7_Templates := "SrcType := Real" } GE_Contact(in1 := #TEOKG1, in2 := 0.0)
      wire#w1
      Contact( #GR1SELP )
      I_Contact( #G2P )
      I_Contact( #G3P )
      I_Contact( #G4P )
      Coil( #G1P )
   END_RUNG
   RUNG wire#w1
      Contact( #GR1SELC1 )
      I_Contact( #G2C1 )
      I_Contact( #G3C1 )
      I_Contact( #G4C1 )
      Coil( #G1C1 )
   END_RUNG
   RUNG wire#w1
      Contact( #GR1SELC2 )
      I_Contact( #G2C2 )
      I_Contact( #G3C2 )
      I_Contact( #G4C2 )
      Coil( #G1C2 )
   END_RUNG
   RUNG wire#w1
      Contact( #GR1SELC3 )
      I_Contact( #G2C3 )
      I_Contact( #G3C3 )
      I_Contact( #G4C3 )
      Coil( #G1C3 )
   END_RUNG
   // the same network as SCL:
   #_w1 := "AlwaysTRUE" AND #G1OK AND (#TEOKG1 >= 0.0);
   #G1P := #_w1 AND #GR1SELP AND NOT #G2P AND NOT #G3P AND NOT #G4P;
   #G1C1 := #_w1 AND #GR1SELC1 AND NOT #G2C1 AND NOT #G3C1 AND NOT #G4C1;
   #G1C2 := #_w1 AND #GR1SELC2 AND NOT #G2C2 AND NOT #G3C2 AND NOT #G4C2;
   #G1C3 := #_w1 AND #GR1SELC3 AND NOT #G2C3 AND NOT #G3C3 AND NOT #G4C3;
END_REGION

REGION Network 50: SELEÇÃO GRUPO 2 COMO PRINCIPAL
   RUNG wire#powerrail
      Contact( "AlwaysTRUE" )
      Contact( #G2OK )
      { S7_Templates := "SrcType := Real" } GE_Contact(in1 := #TEOKG2, in2 := 0.0)
      wire#w1
      Contact( #GR2SELP )
      I_Contact( #G1P )
      I_Contact( #G3P )
      I_Contact( #G4P )
      Coil( #G2P )
   END_RUNG
   RUNG wire#w1
      Contact( #GR2SELC1 )
      I_Contact( #G1C1 )
      I_Contact( #G3C1 )
      I_Contact( #G4C1 )
      Coil( #G2C1 )
   END_RUNG
   RUNG wire#w1
      Contact( #GR2SELC2 )
      I_Contact( #G1C2 )
      I_Contact( #G3C2 )
      I_Contact( #G4C2 )
      Coil( #G2C2 )
   END_RUNG
   RUNG wire#w1
      Contact( #GR2SELC3 )
      I_Contact( #G1C3 )
      I_Contact( #G3C3 )
      I_Contact( #G4C3 )
      Coil( #G2C3 )
   END_RUNG
   // the same network as SCL:
   #_w1 := "AlwaysTRUE" AND #G2OK AND (#TEOKG2 >= 0.0);
   #G2P := #_w1 AND #GR2SELP AND NOT #G1P AND NOT #G3P AND NOT #G4P;
   #G2C1 := #_w1 AND #GR2SELC1 AND NOT #G1C1 AND NOT #G3C1 AND NOT #G4C1;
   #G2C2 := #_w1 AND #GR2SELC2 AND NOT #G1C2 AND NOT #G3C2 AND NOT #G4C2;
   #G2C3 := #_w1 AND #GR2SELC3 AND NOT #G1C3 AND NOT #G3C3 AND NOT #G4C3;
END_REGION

REGION Network 51: SELEÇÃO GRUPO 3 COMO PRINCIPAL
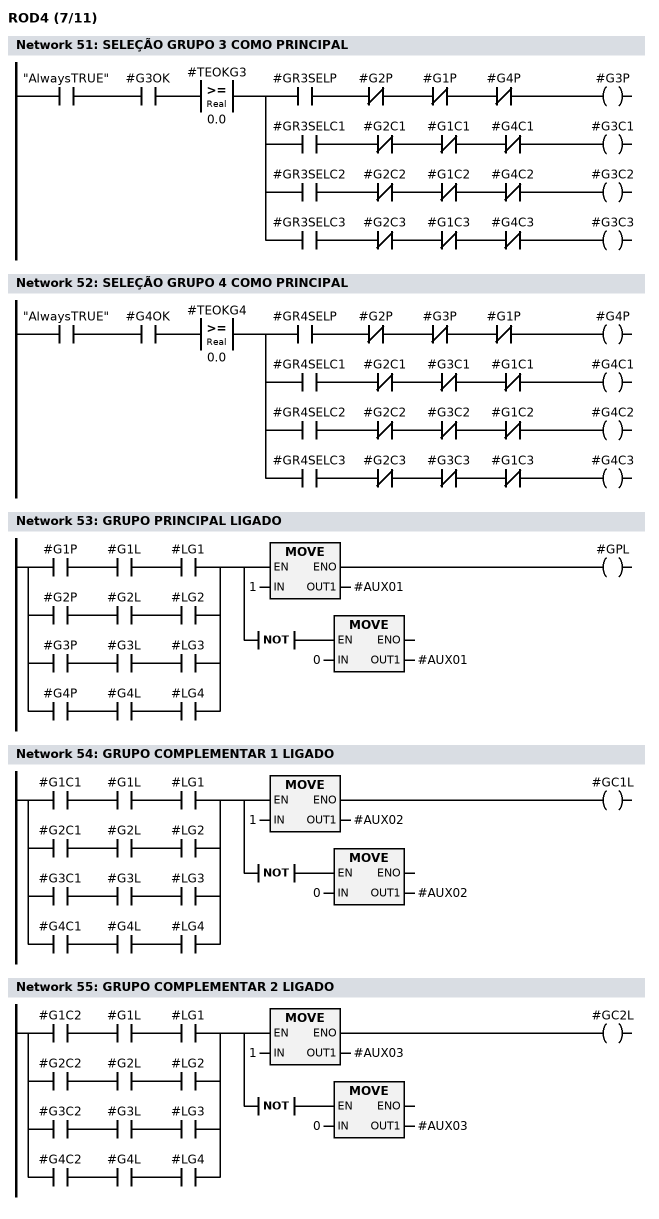
   RUNG wire#powerrail
      Contact( "AlwaysTRUE" )
      Contact( #G3OK )
      { S7_Templates := "SrcType := Real" } GE_Contact(in1 := #TEOKG3, in2 := 0.0)
      wire#w1
      Contact( #GR3SELP )
      I_Contact( #G2P )
      I_Contact( #G1P )
      I_Contact( #G4P )
      Coil( #G3P )
   END_RUNG
   RUNG wire#w1
      Contact( #GR3SELC1 )
      I_Contact( #G2C1 )
      I_Contact( #G1C1 )
      I_Contact( #G4C1 )
      Coil( #G3C1 )
   END_RUNG
   RUNG wire#w1
      Contact( #GR3SELC2 )
      I_Contact( #G2C2 )
      I_Contact( #G1C2 )
      I_Contact( #G4C2 )
      Coil( #G3C2 )
   END_RUNG
   RUNG wire#w1
      Contact( #GR3SELC3 )
      I_Contact( #G2C3 )
      I_Contact( #G1C3 )
      I_Contact( #G4C3 )
      Coil( #G3C3 )
   END_RUNG
   // the same network as SCL:
   #_w1 := "AlwaysTRUE" AND #G3OK AND (#TEOKG3 >= 0.0);
   #G3P := #_w1 AND #GR3SELP AND NOT #G2P AND NOT #G1P AND NOT #G4P;
   #G3C1 := #_w1 AND #GR3SELC1 AND NOT #G2C1 AND NOT #G1C1 AND NOT #G4C1;
   #G3C2 := #_w1 AND #GR3SELC2 AND NOT #G2C2 AND NOT #G1C2 AND NOT #G4C2;
   #G3C3 := #_w1 AND #GR3SELC3 AND NOT #G2C3 AND NOT #G1C3 AND NOT #G4C3;
END_REGION

REGION Network 52: SELEÇÃO GRUPO 4 COMO PRINCIPAL
   RUNG wire#powerrail
      Contact( "AlwaysTRUE" )
      Contact( #G4OK )
      { S7_Templates := "SrcType := Real" } GE_Contact(in1 := #TEOKG4, in2 := 0.0)
      wire#w1
      Contact( #GR4SELP )
      I_Contact( #G2P )
      I_Contact( #G3P )
      I_Contact( #G1P )
      Coil( #G4P )
   END_RUNG
   RUNG wire#w1
      Contact( #GR4SELC1 )
      I_Contact( #G2C1 )
      I_Contact( #G3C1 )
      I_Contact( #G1C1 )
      Coil( #G4C1 )
   END_RUNG
   RUNG wire#w1
      Contact( #GR4SELC2 )
      I_Contact( #G2C2 )
      I_Contact( #G3C2 )
      I_Contact( #G1C2 )
      Coil( #G4C2 )
   END_RUNG
   RUNG wire#w1
      Contact( #GR4SELC3 )
      I_Contact( #G2C3 )
      I_Contact( #G3C3 )
      I_Contact( #G1C3 )
      Coil( #G4C3 )
   END_RUNG
   // the same network as SCL:
   #_w1 := "AlwaysTRUE" AND #G4OK AND (#TEOKG4 >= 0.0);
   #G4P := #_w1 AND #GR4SELP AND NOT #G2P AND NOT #G3P AND NOT #G1P;
   #G4C1 := #_w1 AND #GR4SELC1 AND NOT #G2C1 AND NOT #G3C1 AND NOT #G1C1;
   #G4C2 := #_w1 AND #GR4SELC2 AND NOT #G2C2 AND NOT #G3C2 AND NOT #G1C2;
   #G4C3 := #_w1 AND #GR4SELC3 AND NOT #G2C3 AND NOT #G3C3 AND NOT #G1C3;
END_REGION

REGION Network 53: GRUPO PRINCIPAL LIGADO
   RUNG wire#powerrail
      Contact( #G1P )
      Contact( #G1L )
      Contact( #LG1 )
      wire#w1
      { S7_GenerateENO := "TRUE" } Move(in := 1, out1 => #AUX01)
      Coil( #GPL )
   END_RUNG
   RUNG wire#powerrail
      Contact( #G2P )
      Contact( #G2L )
      Contact( #LG2 )
   END_RUNG wire#w1
   RUNG wire#powerrail
      Contact( #G3P )
      Contact( #G3L )
      Contact( #LG3 )
   END_RUNG wire#w1
   RUNG wire#powerrail
      Contact( #G4P )
      Contact( #G4L )
      Contact( #LG4 )
   END_RUNG wire#w1
   RUNG wire#w1
      Not()
      { S7_GenerateENO := "TRUE" } Move(in := 0, out1 => #AUX01)
   END_RUNG
   // the same network as SCL:
   // ENO of a box is taken as its EN; it also drops when the box reports an error
   #_w1 := (#G1P AND #G1L AND #LG1) OR (#G2P AND #G2L AND #LG2) OR (#G3P AND #G3L AND #LG3) OR (#G4P AND #G4L AND #LG4);
   IF #_w1 THEN #AUX01 := 1; END_IF;
   #GPL := #_w1;
   IF NOT #_w1 THEN #AUX01 := 0; END_IF;
END_REGION

REGION Network 54: GRUPO COMPLEMENTAR 1 LIGADO
   RUNG wire#powerrail
      Contact( #G1C1 )
      Contact( #G1L )
      Contact( #LG1 )
      wire#w1
      { S7_GenerateENO := "TRUE" } Move(in := 1, out1 => #AUX02)
      Coil( #GC1L )
   END_RUNG
   RUNG wire#powerrail
      Contact( #G2C1 )
      Contact( #G2L )
      Contact( #LG2 )
   END_RUNG wire#w1
   RUNG wire#powerrail
      Contact( #G3C1 )
      Contact( #G3L )
      Contact( #LG3 )
   END_RUNG wire#w1
   RUNG wire#powerrail
      Contact( #G4C1 )
      Contact( #G4L )
      Contact( #LG4 )
   END_RUNG wire#w1
   RUNG wire#w1
      Not()
      { S7_GenerateENO := "TRUE" } Move(in := 0, out1 => #AUX02)
   END_RUNG
   // the same network as SCL:
   // ENO of a box is taken as its EN; it also drops when the box reports an error
   #_w1 := (#G1C1 AND #G1L AND #LG1) OR (#G2C1 AND #G2L AND #LG2) OR (#G3C1 AND #G3L AND #LG3) OR (#G4C1 AND #G4L AND #LG4);
   IF #_w1 THEN #AUX02 := 1; END_IF;
   #GC1L := #_w1;
   IF NOT #_w1 THEN #AUX02 := 0; END_IF;
END_REGION

REGION Network 55: GRUPO COMPLEMENTAR 2 LIGADO
   RUNG wire#powerrail
      Contact( #G1C2 )
      Contact( #G1L )
      Contact( #LG1 )
      wire#w1
      { S7_GenerateENO := "TRUE" } Move(in := 1, out1 => #AUX03)
      Coil( #GC2L )
   END_RUNG
   RUNG wire#powerrail
      Contact( #G2C2 )
      Contact( #G2L )
      Contact( #LG2 )
   END_RUNG wire#w1
   RUNG wire#powerrail
      Contact( #G3C2 )
      Contact( #G3L )
      Contact( #LG3 )
   END_RUNG wire#w1
   RUNG wire#powerrail
      Contact( #G4C2 )
      Contact( #G4L )
      Contact( #LG4 )
   END_RUNG wire#w1
   RUNG wire#w1
      Not()
      { S7_GenerateENO := "TRUE" } Move(in := 0, out1 => #AUX03)
   END_RUNG
   // the same network as SCL:
   // ENO of a box is taken as its EN; it also drops when the box reports an error
   #_w1 := (#G1C2 AND #G1L AND #LG1) OR (#G2C2 AND #G2L AND #LG2) OR (#G3C2 AND #G3L AND #LG3) OR (#G4C2 AND #G4L AND #LG4);
   IF #_w1 THEN #AUX03 := 1; END_IF;
   #GC2L := #_w1;
   IF NOT #_w1 THEN #AUX03 := 0; END_IF;
END_REGION

REGION Network 56: GRUPO COMPLEMENTAR 3 LIGADO
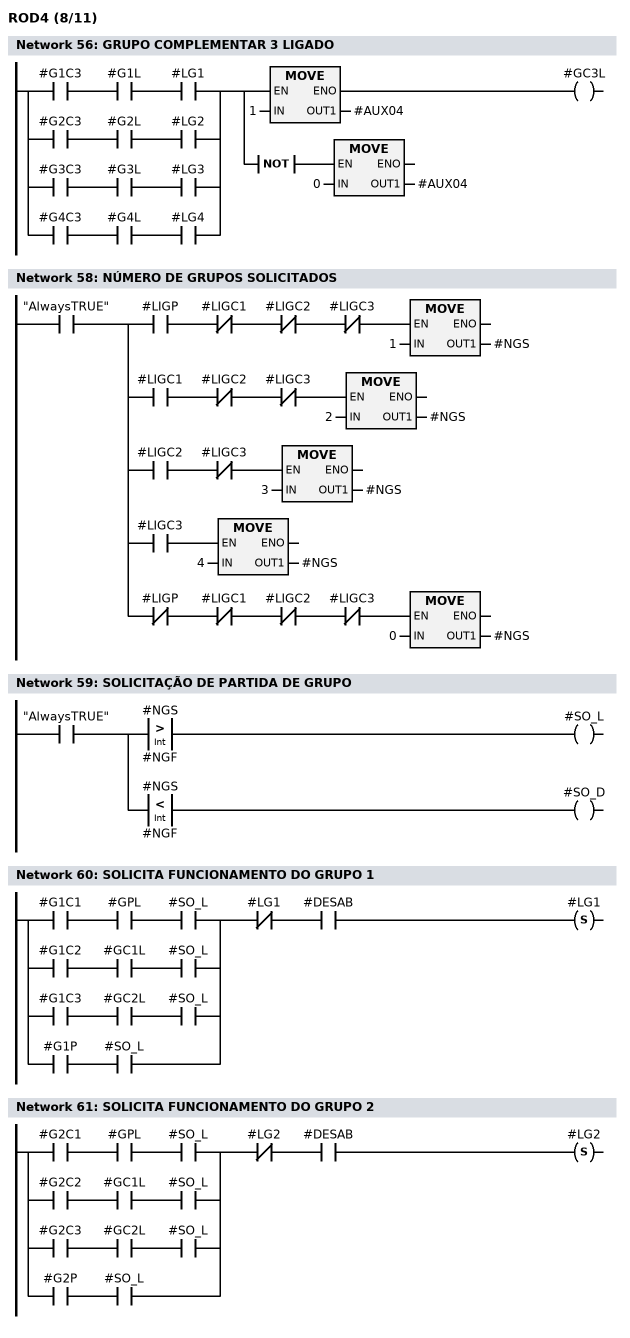
   RUNG wire#powerrail
      Contact( #G1C3 )
      Contact( #G1L )
      Contact( #LG1 )
      wire#w1
      { S7_GenerateENO := "TRUE" } Move(in := 1, out1 => #AUX04)
      Coil( #GC3L )
   END_RUNG
   RUNG wire#powerrail
      Contact( #G2C3 )
      Contact( #G2L )
      Contact( #LG2 )
   END_RUNG wire#w1
   RUNG wire#powerrail
      Contact( #G3C3 )
      Contact( #G3L )
      Contact( #LG3 )
   END_RUNG wire#w1
   RUNG wire#powerrail
      Contact( #G4C3 )
      Contact( #G4L )
      Contact( #LG4 )
   END_RUNG wire#w1
   RUNG wire#w1
      Not()
      { S7_GenerateENO := "TRUE" } Move(in := 0, out1 => #AUX04)
   END_RUNG
   // the same network as SCL:
   // ENO of a box is taken as its EN; it also drops when the box reports an error
   #_w1 := (#G1C3 AND #G1L AND #LG1) OR (#G2C3 AND #G2L AND #LG2) OR (#G3C3 AND #G3L AND #LG3) OR (#G4C3 AND #G4L AND #LG4);
   IF #_w1 THEN #AUX04 := 1; END_IF;
   #GC3L := #_w1;
   IF NOT #_w1 THEN #AUX04 := 0; END_IF;
END_REGION

NETWORK
TITLE = NÚMERO DE GRUPOS FUNCIONANDO

      L     #AUX01;
      L     #AUX02;
      +I;
      L     #AUX03;
      +I;
      L     #AUX04;
      +I;
      T     #NGF;

REGION Network 58: NÚMERO DE GRUPOS SOLICITADOS
   RUNG wire#powerrail
      Contact( "AlwaysTRUE" )
      wire#w1
      Contact( #LIGP )
      I_Contact( #LIGC1 )
      I_Contact( #LIGC2 )
      I_Contact( #LIGC3 )
      { S7_GenerateENO := "TRUE" } Move(in := 1, out1 => #NGS)
   END_RUNG
   RUNG wire#w1
      Contact( #LIGC1 )
      I_Contact( #LIGC2 )
      I_Contact( #LIGC3 )
      { S7_GenerateENO := "TRUE" } Move(in := 2, out1 => #NGS)
   END_RUNG
   RUNG wire#w1
      Contact( #LIGC2 )
      I_Contact( #LIGC3 )
      { S7_GenerateENO := "TRUE" } Move(in := 3, out1 => #NGS)
   END_RUNG
   RUNG wire#w1
      Contact( #LIGC3 )
      { S7_GenerateENO := "TRUE" } Move(in := 4, out1 => #NGS)
   END_RUNG
   RUNG wire#w1
      I_Contact( #LIGP )
      I_Contact( #LIGC1 )
      I_Contact( #LIGC2 )
      I_Contact( #LIGC3 )
      { S7_GenerateENO := "TRUE" } Move(in := 0, out1 => #NGS)
   END_RUNG
   // the same network as SCL:
   IF "AlwaysTRUE" AND #LIGP AND NOT #LIGC1 AND NOT #LIGC2 AND NOT #LIGC3 THEN #NGS := 1; END_IF;
   IF "AlwaysTRUE" AND #LIGC1 AND NOT #LIGC2 AND NOT #LIGC3 THEN #NGS := 2; END_IF;
   IF "AlwaysTRUE" AND #LIGC2 AND NOT #LIGC3 THEN #NGS := 3; END_IF;
   IF "AlwaysTRUE" AND #LIGC3 THEN #NGS := 4; END_IF;
   IF "AlwaysTRUE" AND NOT #LIGP AND NOT #LIGC1 AND NOT #LIGC2 AND NOT #LIGC3 THEN #NGS := 0; END_IF;
END_REGION

REGION Network 59: SOLICITAÇÃO DE PARTIDA DE GRUPO
   RUNG wire#powerrail
      Contact( "AlwaysTRUE" )
      wire#w1
      { S7_Templates := "SrcType := Int" } GT_Contact(in1 := #NGS, in2 := #NGF)
      Coil( #SO_L )
   END_RUNG
   RUNG wire#w1
      { S7_Templates := "SrcType := Int" } LT_Contact(in1 := #NGS, in2 := #NGF)
      Coil( #SO_D )
   END_RUNG
   // the same network as SCL:
   #SO_L := "AlwaysTRUE" AND (#NGS > #NGF);
   #SO_D := "AlwaysTRUE" AND (#NGS < #NGF);
END_REGION

REGION Network 60: SOLICITA FUNCIONAMENTO DO GRUPO 1
   RUNG wire#powerrail
      Contact( #G1C1 )
      Contact( #GPL )
      Contact( #SO_L )
      wire#w1
      I_Contact( #LG1 )
      Contact( #DESAB )
      S_Coil( #LG1 )
   END_RUNG
   RUNG wire#powerrail
      Contact( #G1C2 )
      Contact( #GC1L )
      Contact( #SO_L )
   END_RUNG wire#w1
   RUNG wire#powerrail
      Contact( #G1C3 )
      Contact( #GC2L )
      Contact( #SO_L )
   END_RUNG wire#w1
   RUNG wire#powerrail
      Contact( #G1P )
      Contact( #SO_L )
   END_RUNG wire#w1
   // the same network as SCL:
   IF ((#G1C1 AND #GPL AND #SO_L) OR (#G1C2 AND #GC1L AND #SO_L) OR (#G1C3 AND #GC2L AND #SO_L) OR (#G1P AND #SO_L)) AND NOT #LG1 AND #DESAB THEN
       #LG1 := TRUE;
   END_IF;
END_REGION

REGION Network 61: SOLICITA FUNCIONAMENTO DO GRUPO 2
   RUNG wire#powerrail
      Contact( #G2C1 )
      Contact( #GPL )
      Contact( #SO_L )
      wire#w1
      I_Contact( #LG2 )
      Contact( #DESAB )
      S_Coil( #LG2 )
   END_RUNG
   RUNG wire#powerrail
      Contact( #G2C2 )
      Contact( #GC1L )
      Contact( #SO_L )
   END_RUNG wire#w1
   RUNG wire#powerrail
      Contact( #G2C3 )
      Contact( #GC2L )
      Contact( #SO_L )
   END_RUNG wire#w1
   RUNG wire#powerrail
      Contact( #G2P )
      Contact( #SO_L )
   END_RUNG wire#w1
   // the same network as SCL:
   IF ((#G2C1 AND #GPL AND #SO_L) OR (#G2C2 AND #GC1L AND #SO_L) OR (#G2C3 AND #GC2L AND #SO_L) OR (#G2P AND #SO_L)) AND NOT #LG2 AND #DESAB THEN
       #LG2 := TRUE;
   END_IF;
END_REGION

REGION Network 62: SOLICITA FUNCIONAMENTO DO GRUPO 3
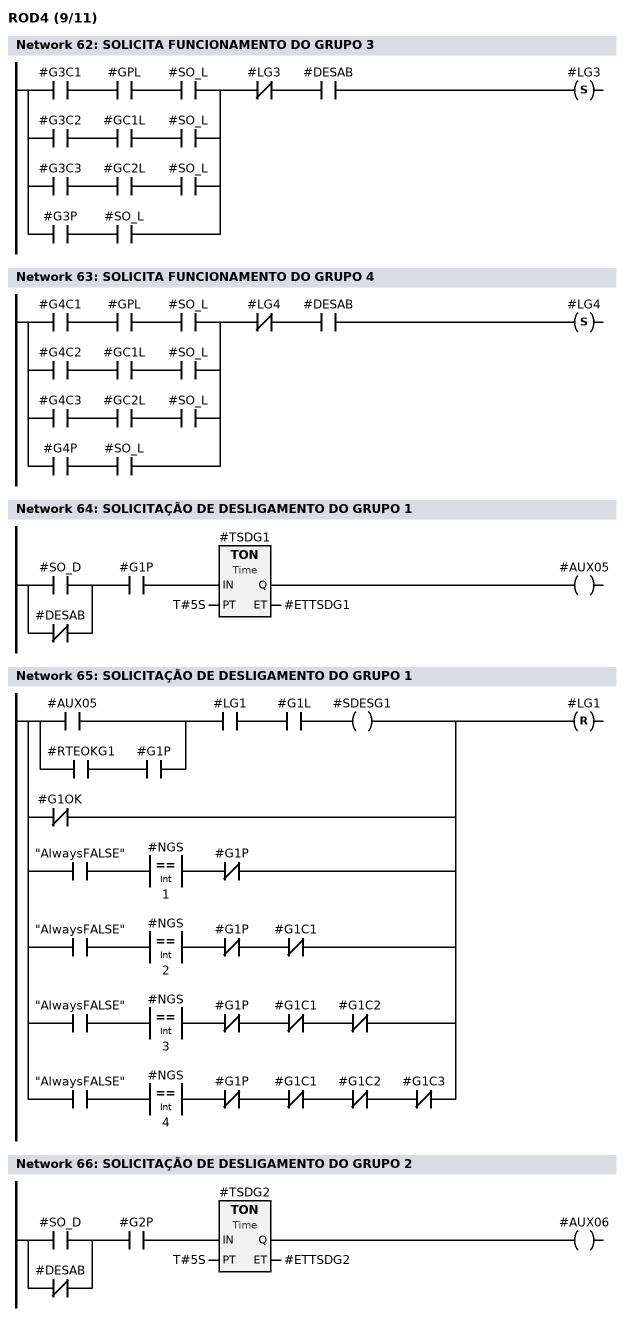
   RUNG wire#powerrail
      Contact( #G3C1 )
      Contact( #GPL )
      Contact( #SO_L )
      wire#w1
      I_Contact( #LG3 )
      Contact( #DESAB )
      S_Coil( #LG3 )
   END_RUNG
   RUNG wire#powerrail
      Contact( #G3C2 )
      Contact( #GC1L )
      Contact( #SO_L )
   END_RUNG wire#w1
   RUNG wire#powerrail
      Contact( #G3C3 )
      Contact( #GC2L )
      Contact( #SO_L )
   END_RUNG wire#w1
   RUNG wire#powerrail
      Contact( #G3P )
      Contact( #SO_L )
   END_RUNG wire#w1
   // the same network as SCL:
   IF ((#G3C1 AND #GPL AND #SO_L) OR (#G3C2 AND #GC1L AND #SO_L) OR (#G3C3 AND #GC2L AND #SO_L) OR (#G3P AND #SO_L)) AND NOT #LG3 AND #DESAB THEN
       #LG3 := TRUE;
   END_IF;
END_REGION

REGION Network 63: SOLICITA FUNCIONAMENTO DO GRUPO 4
   RUNG wire#powerrail
      Contact( #G4C1 )
      Contact( #GPL )
      Contact( #SO_L )
      wire#w1
      I_Contact( #LG4 )
      Contact( #DESAB )
      S_Coil( #LG4 )
   END_RUNG
   RUNG wire#powerrail
      Contact( #G4C2 )
      Contact( #GC1L )
      Contact( #SO_L )
   END_RUNG wire#w1
   RUNG wire#powerrail
      Contact( #G4C3 )
      Contact( #GC2L )
      Contact( #SO_L )
   END_RUNG wire#w1
   RUNG wire#powerrail
      Contact( #G4P )
      Contact( #SO_L )
   END_RUNG wire#w1
   // the same network as SCL:
   IF ((#G4C1 AND #GPL AND #SO_L) OR (#G4C2 AND #GC1L AND #SO_L) OR (#G4C3 AND #GC2L AND #SO_L) OR (#G4P AND #SO_L)) AND NOT #LG4 AND #DESAB THEN
       #LG4 := TRUE;
   END_IF;
END_REGION

REGION Network 64: SOLICITAÇÃO DE DESLIGAMENTO DO GRUPO 1
   RUNG wire#powerrail
      Contact( #SO_D )
      wire#w1
      Contact( #G1P )
      { S7_Templates := "time_type := Time" } #TSDG1.TON(pt := T#5S, et => #ETTSDG1)
      Coil( #AUX05 )
   END_RUNG
   RUNG wire#powerrail
      I_Contact( #DESAB )
   END_RUNG wire#w1
   // the same network as SCL:
   #TSDG1(IN := (#SO_D OR NOT #DESAB) AND #G1P, PT := T#5S, ET => #ETTSDG1);   // TON
   #AUX05 := #TSDG1.Q;
END_REGION

REGION Network 65: SOLICITAÇÃO DE DESLIGAMENTO DO GRUPO 1
   RUNG wire#powerrail
      Contact( #AUX05 )
      wire#w1
      Contact( #LG1 )
      Contact( #G1L )
      Coil( #SDESG1 )
      wire#w2
      R_Coil( #LG1 )
   END_RUNG
   RUNG wire#powerrail
      Contact( #RTEOKG1 )
      Contact( #G1P )
   END_RUNG wire#w1
   RUNG wire#powerrail
      I_Contact( #G1OK )
   END_RUNG wire#w2
   RUNG wire#powerrail
      Contact( "AlwaysFALSE" )
      { S7_Templates := "SrcType := Int" } EQ_Contact(in1 := #NGS, in2 := 1)
      I_Contact( #G1P )
   END_RUNG wire#w2
   RUNG wire#powerrail
      Contact( "AlwaysFALSE" )
      { S7_Templates := "SrcType := Int" } EQ_Contact(in1 := #NGS, in2 := 2)
      I_Contact( #G1P )
      I_Contact( #G1C1 )
   END_RUNG wire#w2
   RUNG wire#powerrail
      Contact( "AlwaysFALSE" )
      { S7_Templates := "SrcType := Int" } EQ_Contact(in1 := #NGS, in2 := 3)
      I_Contact( #G1P )
      I_Contact( #G1C1 )
      I_Contact( #G1C2 )
   END_RUNG wire#w2
   RUNG wire#powerrail
      Contact( "AlwaysFALSE" )
      { S7_Templates := "SrcType := Int" } EQ_Contact(in1 := #NGS, in2 := 4)
      I_Contact( #G1P )
      I_Contact( #G1C1 )
      I_Contact( #G1C2 )
      I_Contact( #G1C3 )
   END_RUNG wire#w2
   // the same network as SCL:
   #SDESG1 := (#AUX05 OR (#RTEOKG1 AND #G1P)) AND #LG1 AND #G1L;
   IF #SDESG1 OR NOT #G1OK OR ("AlwaysFALSE" AND (#NGS = 1) AND NOT #G1P) OR ("AlwaysFALSE" AND (#NGS = 2) AND NOT #G1P AND NOT #G1C1) OR ("AlwaysFALSE" AND (#NGS = 3) AND NOT #G1P AND NOT #G1C1 AND NOT #G1C2) OR ("AlwaysFALSE" AND (#NGS = 4) AND NOT #G1P AND NOT #G1C1 AND NOT #G1C2 AND NOT #G1C3) THEN
       #LG1 := FALSE;
   END_IF;
END_REGION

REGION Network 66: SOLICITAÇÃO DE DESLIGAMENTO DO GRUPO 2
   RUNG wire#powerrail
      Contact( #SO_D )
      wire#w1
      Contact( #G2P )
      { S7_Templates := "time_type := Time" } #TSDG2.TON(pt := T#5S, et => #ETTSDG2)
      Coil( #AUX06 )
   END_RUNG
   RUNG wire#powerrail
      I_Contact( #DESAB )
   END_RUNG wire#w1
   // the same network as SCL:
   #TSDG2(IN := (#SO_D OR NOT #DESAB) AND #G2P, PT := T#5S, ET => #ETTSDG2);   // TON
   #AUX06 := #TSDG2.Q;
END_REGION

REGION Network 67: SOLICITAÇÃO DE DESLIGAMENTO DO GRUPO 2
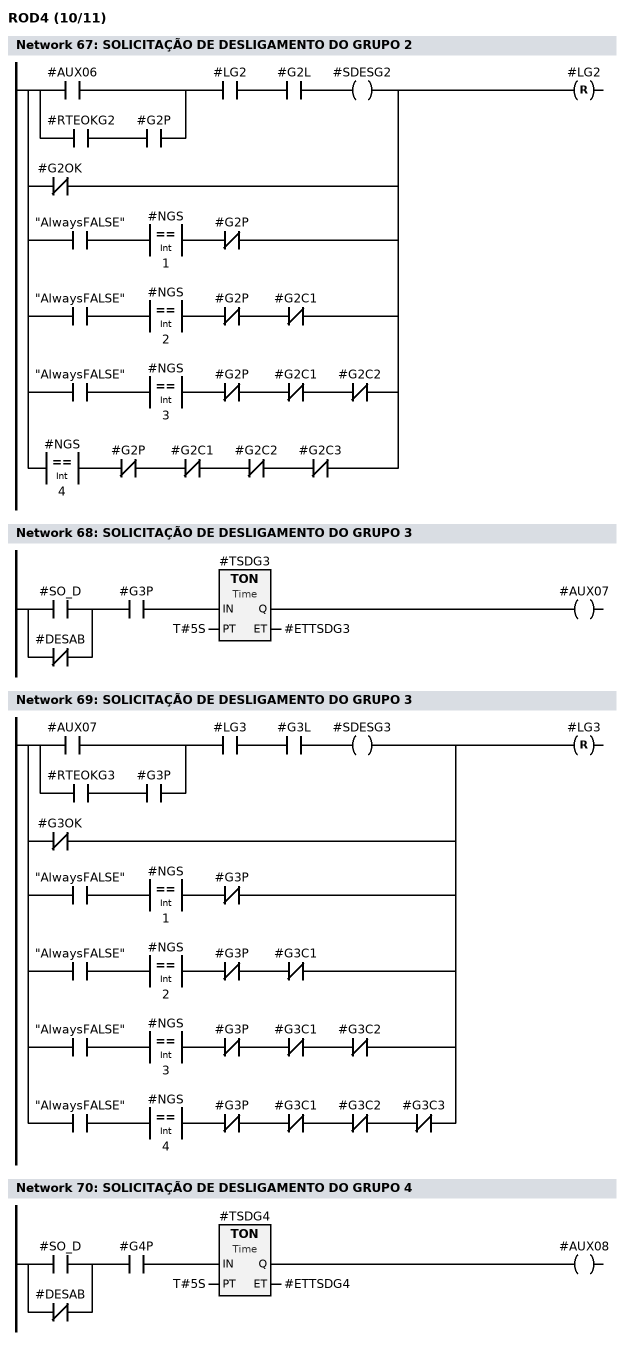
   RUNG wire#powerrail
      Contact( #AUX06 )
      wire#w1
      Contact( #LG2 )
      Contact( #G2L )
      Coil( #SDESG2 )
      wire#w2
      R_Coil( #LG2 )
   END_RUNG
   RUNG wire#powerrail
      Contact( #RTEOKG2 )
      Contact( #G2P )
   END_RUNG wire#w1
   RUNG wire#powerrail
      I_Contact( #G2OK )
   END_RUNG wire#w2
   RUNG wire#powerrail
      Contact( "AlwaysFALSE" )
      { S7_Templates := "SrcType := Int" } EQ_Contact(in1 := #NGS, in2 := 1)
      I_Contact( #G2P )
   END_RUNG wire#w2
   RUNG wire#powerrail
      Contact( "AlwaysFALSE" )
      { S7_Templates := "SrcType := Int" } EQ_Contact(in1 := #NGS, in2 := 2)
      I_Contact( #G2P )
      I_Contact( #G2C1 )
   END_RUNG wire#w2
   RUNG wire#powerrail
      Contact( "AlwaysFALSE" )
      { S7_Templates := "SrcType := Int" } EQ_Contact(in1 := #NGS, in2 := 3)
      I_Contact( #G2P )
      I_Contact( #G2C1 )
      I_Contact( #G2C2 )
   END_RUNG wire#w2
   RUNG wire#powerrail
      { S7_Templates := "SrcType := Int" } EQ_Contact(in1 := #NGS, in2 := 4)
      I_Contact( #G2P )
      I_Contact( #G2C1 )
      I_Contact( #G2C2 )
      I_Contact( #G2C3 )
   END_RUNG wire#w2
   // the same network as SCL:
   #SDESG2 := (#AUX06 OR (#RTEOKG2 AND #G2P)) AND #LG2 AND #G2L;
   IF #SDESG2 OR NOT #G2OK OR ("AlwaysFALSE" AND (#NGS = 1) AND NOT #G2P) OR ("AlwaysFALSE" AND (#NGS = 2) AND NOT #G2P AND NOT #G2C1) OR ("AlwaysFALSE" AND (#NGS = 3) AND NOT #G2P AND NOT #G2C1 AND NOT #G2C2) OR ((#NGS = 4) AND NOT #G2P AND NOT #G2C1 AND NOT #G2C2 AND NOT #G2C3) THEN
       #LG2 := FALSE;
   END_IF;
END_REGION

REGION Network 68: SOLICITAÇÃO DE DESLIGAMENTO DO GRUPO 3
   RUNG wire#powerrail
      Contact( #SO_D )
      wire#w1
      Contact( #G3P )
      { S7_Templates := "time_type := Time" } #TSDG3.TON(pt := T#5S, et => #ETTSDG3)
      Coil( #AUX07 )
   END_RUNG
   RUNG wire#powerrail
      I_Contact( #DESAB )
   END_RUNG wire#w1
   // the same network as SCL:
   #TSDG3(IN := (#SO_D OR NOT #DESAB) AND #G3P, PT := T#5S, ET => #ETTSDG3);   // TON
   #AUX07 := #TSDG3.Q;
END_REGION

REGION Network 69: SOLICITAÇÃO DE DESLIGAMENTO DO GRUPO 3
   RUNG wire#powerrail
      Contact( #AUX07 )
      wire#w1
      Contact( #LG3 )
      Contact( #G3L )
      Coil( #SDESG3 )
      wire#w2
      R_Coil( #LG3 )
   END_RUNG
   RUNG wire#powerrail
      Contact( #RTEOKG3 )
      Contact( #G3P )
   END_RUNG wire#w1
   RUNG wire#powerrail
      I_Contact( #G3OK )
   END_RUNG wire#w2
   RUNG wire#powerrail
      Contact( "AlwaysFALSE" )
      { S7_Templates := "SrcType := Int" } EQ_Contact(in1 := #NGS, in2 := 1)
      I_Contact( #G3P )
   END_RUNG wire#w2
   RUNG wire#powerrail
      Contact( "AlwaysFALSE" )
      { S7_Templates := "SrcType := Int" } EQ_Contact(in1 := #NGS, in2 := 2)
      I_Contact( #G3P )
      I_Contact( #G3C1 )
   END_RUNG wire#w2
   RUNG wire#powerrail
      Contact( "AlwaysFALSE" )
      { S7_Templates := "SrcType := Int" } EQ_Contact(in1 := #NGS, in2 := 3)
      I_Contact( #G3P )
      I_Contact( #G3C1 )
      I_Contact( #G3C2 )
   END_RUNG wire#w2
   RUNG wire#powerrail
      Contact( "AlwaysFALSE" )
      { S7_Templates := "SrcType := Int" } EQ_Contact(in1 := #NGS, in2 := 4)
      I_Contact( #G3P )
      I_Contact( #G3C1 )
      I_Contact( #G3C2 )
      I_Contact( #G3C3 )
   END_RUNG wire#w2
   // the same network as SCL:
   #SDESG3 := (#AUX07 OR (#RTEOKG3 AND #G3P)) AND #LG3 AND #G3L;
   IF #SDESG3 OR NOT #G3OK OR ("AlwaysFALSE" AND (#NGS = 1) AND NOT #G3P) OR ("AlwaysFALSE" AND (#NGS = 2) AND NOT #G3P AND NOT #G3C1) OR ("AlwaysFALSE" AND (#NGS = 3) AND NOT #G3P AND NOT #G3C1 AND NOT #G3C2) OR ("AlwaysFALSE" AND (#NGS = 4) AND NOT #G3P AND NOT #G3C1 AND NOT #G3C2 AND NOT #G3C3) THEN
       #LG3 := FALSE;
   END_IF;
END_REGION

REGION Network 70: SOLICITAÇÃO DE DESLIGAMENTO DO GRUPO 4
   RUNG wire#powerrail
      Contact( #SO_D )
      wire#w1
      Contact( #G4P )
      { S7_Templates := "time_type := Time" } #TSDG4.TON(pt := T#5S, et => #ETTSDG4)
      Coil( #AUX08 )
   END_RUNG
   RUNG wire#powerrail
      I_Contact( #DESAB )
   END_RUNG wire#w1
   // the same network as SCL:
   #TSDG4(IN := (#SO_D OR NOT #DESAB) AND #G4P, PT := T#5S, ET => #ETTSDG4);   // TON
   #AUX08 := #TSDG4.Q;
END_REGION

REGION Network 71: SOLICITAÇÃO DE DESLIGAMENTO DO GRUPO 4
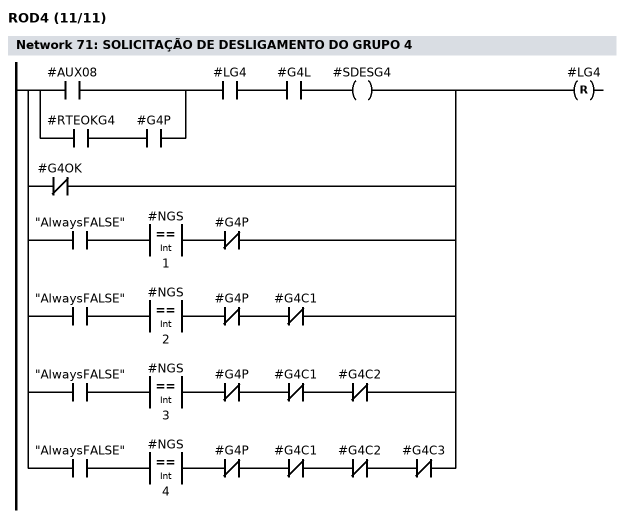
   RUNG wire#powerrail
      Contact( #AUX08 )
      wire#w1
      Contact( #LG4 )
      Contact( #G4L )
      Coil( #SDESG4 )
      wire#w2
      R_Coil( #LG4 )
   END_RUNG
   RUNG wire#powerrail
      Contact( #RTEOKG4 )
      Contact( #G4P )
   END_RUNG wire#w1
   RUNG wire#powerrail
      I_Contact( #G4OK )
   END_RUNG wire#w2
   RUNG wire#powerrail
      Contact( "AlwaysFALSE" )
      { S7_Templates := "SrcType := Int" } EQ_Contact(in1 := #NGS, in2 := 1)
      I_Contact( #G4P )
   END_RUNG wire#w2
   RUNG wire#powerrail
      Contact( "AlwaysFALSE" )
      { S7_Templates := "SrcType := Int" } EQ_Contact(in1 := #NGS, in2 := 2)
      I_Contact( #G4P )
      I_Contact( #G4C1 )
   END_RUNG wire#w2
   RUNG wire#powerrail
      Contact( "AlwaysFALSE" )
      { S7_Templates := "SrcType := Int" } EQ_Contact(in1 := #NGS, in2 := 3)
      I_Contact( #G4P )
      I_Contact( #G4C1 )
      I_Contact( #G4C2 )
   END_RUNG wire#w2
   RUNG wire#powerrail
      Contact( "AlwaysFALSE" )
      { S7_Templates := "SrcType := Int" } EQ_Contact(in1 := #NGS, in2 := 4)
      I_Contact( #G4P )
      I_Contact( #G4C1 )
      I_Contact( #G4C2 )
      I_Contact( #G4C3 )
   END_RUNG wire#w2
   // the same network as SCL:
   #SDESG4 := (#AUX08 OR (#RTEOKG4 AND #G4P)) AND #LG4 AND #G4L;
   IF #SDESG4 OR NOT #G4OK OR ("AlwaysFALSE" AND (#NGS = 1) AND NOT #G4P) OR ("AlwaysFALSE" AND (#NGS = 2) AND NOT #G4P AND NOT #G4C1) OR ("AlwaysFALSE" AND (#NGS = 3) AND NOT #G4P AND NOT #G4C1 AND NOT #G4C2) OR ("AlwaysFALSE" AND (#NGS = 4) AND NOT #G4P AND NOT #G4C1 AND NOT #G4C2 AND NOT #G4C3) THEN
       #LG4 := FALSE;
   END_IF;
END_REGION
END_FUNCTION_BLOCK
